TYPE ST_ServoInterlocks :
STRUCT
	Move_Positive : BOOL;
	Move_Negative : BOOL;
	SafetyOk     : BOOL;
	
END_STRUCT
END_TYPE

(* stored: Version 1.1.0.1, ProductVersion 3.1.4024.12
   DUT ST_ServoInterlocks: Id {07679274-de7f-4bf4-ac09-4ebdcd9540a1} *)
